{attribute addProperty BoxType "EL3692-0000-0017"}
{attribute addProperty Id "SAI_Inputs_Channel_1AT %I*SAI_Inputs_Channel_64E745974860SAI_Range_Channel_1AT %I*SAI_Range_Channel_DF9848341620SAI_Inputs_Real_Channel_1AT %I*SAI_Inputs_Real_Channel_5F0304D13240SAI_Inputs_Channel_2AT %I*SAI_Inputs_Channel_64E745974860SAI_Range_Channel_2AT %I*SAI_Range_Channel_DF9848341620SAI_Inputs_Real_Channel_2AT %I*SAI_Inputs_Real_Channel_5F0304D13240WcStateAT %I*WcState_98A4DF7520.250InfoDataAT %I*InfoData_BC63D37F80100"}
{attribute addProperty CRC "3877237170"}
{attribute addProperty SizeInBites "274"}
{attribute addProperty SizeInBytes "34.25"}
TYPE EL3692_04436164 :
STRUCT
	{attribute addProperty Name "SAI_Inputs_Channel_1"}
	SAI_Inputs_Channel_1 : SAI_Inputs_Channel_64E74597;
	{attribute addProperty Name "SAI_Range_Channel_1"}
	SAI_Range_Channel_1 : SAI_Range_Channel_DF984834;
	{attribute addProperty Name "SAI_Inputs_Real_Channel_1"}
	SAI_Inputs_Real_Channel_1 : SAI_Inputs_Real_Channel_5F0304D1;
	{attribute addProperty Name "SAI_Inputs_Channel_2"}
	SAI_Inputs_Channel_2 : SAI_Inputs_Channel_64E74597;
	{attribute addProperty Name "SAI_Range_Channel_2"}
	SAI_Range_Channel_2 : SAI_Range_Channel_DF984834;
	{attribute addProperty Name "SAI_Inputs_Real_Channel_2"}
	SAI_Inputs_Real_Channel_2 : SAI_Inputs_Real_Channel_5F0304D1;
	{attribute addProperty Name "WcState"}
	WcState : WcState_98A4DF75;
	{attribute addProperty Name "InfoData"}
	InfoData : InfoData_BC63D37F;
END_STRUCT
END_TYPE

(* stored: Version 1.2.0.0, ProductVersion 3.1.4024.9
   DUT EL3692_04436164: Id {942c63c2-801c-44a2-a238-c7755d1bec57} *)
